// TwinCAT 3 PLC project SFICrane
// ProgramVersion: 3.1.4023.0
// libraries:
//   Tc2_MC2, * (Beckhoff Automation GmbH)
//   Tc2_MC2_Drive, * (Beckhoff Automation GmbH)
//   Tc2_Standard, * (Beckhoff Automation GmbH)
//   Tc2_System, * (Beckhoff Automation GmbH)
//   Tc2_Utilities, * (Beckhoff Automation GmbH)
//   Tc3_Module, * (Beckhoff Automation GmbH)
// project tree:
//   AXIS CONTROL/ GVL_AXIS1.TcGVL, GVL_AXIS2.TcGVL (not stored), GVL_AXIS3.TcGVL, GVL_AXIS4.TcGVL (not stored), GVL_Safety_AXIS4.TcGVL (not stored), GVL_Safety_IO.TcGVL, P_AxisControl.TcPOU, ST_MC_CMD.TcDUT, ST_MC_ParametersAxis.TcDUT, ST_MC_Status.TcDUT (not stored)
//   INPUTS/Function Blocks/ FB_AnalogInputScaling.TcPOU, FB_JoystickInputScaling.TcPOU
//   INPUTS/ G_Inputs.TcGVL, G_Sensors.TcGVL (not stored), P_Inputs.TcPOU (not stored)
//   INPUTS/Struct/ ST_AnalogInput.TcDUT (not stored), ST_AnalogInputScaling.TcDUT (not stored), ST_AnalogInputStatus.TcDUT, ST_JoystickInputScaling.TcDUT (not stored)
//   MACHINE CONTROL/ G_Parameters.TcGVL, G_Work.TcGVL (not stored), P_MachineControl.TcPOU
//   MACHINE CONTROL/InverseKinematics2d/ cosd.TcPOU (not stored), FB_InverseKin2d.TcPOU (not stored), GVL_InverseKinematics.TcGVL (not stored), rt_ceild.TcPOU (not stored), rt_floord.TcPOU, rt_remd.TcPOU (not stored)
//   MACHINE CONTROL/Struct/ ST_Parameters.TcDUT (not stored)
//   OUTPUTS/ G_Outputs.TcGVL (not stored), P_Outputs.TcPOU (not stored)
//   / PlcTask.TcTTO
//   POUs/ MAIN.TcPOU
// real-time tasks:
//   TASK PlcTask: cycle T#10ms, priority 20, ADS port 350
// motion (NC):
//   TASK NC-Task 1 SAF: cycle T#2ms, priority 4, ADS port 501
//   TASK NC-Task 1 SVB: cycle T#10ms, priority 8, ADS port 511
//   AXIS Axis 1 - Bottom cylinder (id 1)
//     OtherSettings: AllowMotionCmdToSlave=true
//     encoder EncType=8
//       EncPara: MaxCount=#x0036ee7f
//     drive DrvType=9
//       DrvPara: MaxCount=#xffffffff, DriveControlDWord=#x00030000
//         Analog: VeloScale=6, TorqueSetpointScale=10, ScaleFactorActTorque=0.1
//         TimeComp: TaskDelayCycles=1
//     controller CtrType=1
//       CtrPara: PriorControlFactor=1
//         Observer: BandWidth=20
//   AXIS Axis 2 - Slew motor (id 2)
//     OtherSettings: AllowMotionCmdToSlave=true
//     encoder EncType=8
//       EncPara: MaxCount=#x0036ee7f
//     drive DrvType=9
//       DrvPara: MaxCount=#xffffffff, DriveControlDWord=#x00030000
//         Analog: VeloScale=6, TorqueSetpointScale=10, ScaleFactorActTorque=0.1
//         TimeComp: TaskDelayCycles=1
//     controller CtrType=1
//       CtrPara: PriorControlFactor=1
//         Observer: BandWidth=20
//   AXIS Axis 3 - Top cylinder (id 3)
//     OtherSettings: AllowMotionCmdToSlave=true
//     encoder EncType=8
//       EncPara: MaxCount=#x0036ee7f
//     drive DrvType=9
//       DrvPara: MaxCount=#xffffffff, DriveControlDWord=#x00030000
//         Analog: VeloScale=6, TorqueSetpointScale=10, ScaleFactorActTorque=0.1
//         TimeComp: TaskDelayCycles=1
//     controller CtrType=1
//       CtrPara: PriorControlFactor=1
//         Observer: BandWidth=20
//   AXIS Axis 4 - Winch motor (id 4)
//     OtherSettings: AllowMotionCmdToSlave=true
//     encoder EncType=19
//       EncPara: MaxCount=#xffffffff
//     drive DrvType=16
//       DrvPara: MaxCount=#xffffffff, DriveControlDWord=#x00020100
//         Analog: TorqueSetpointScale=10, ScaleFactorActTorque=0.1
//         TimeComp: TaskDelayCycles=1
//     controller CtrType=1
//       CtrPara: PriorControlFactor=1
//         Observer: BandWidth=20
// I/O:
//   DEVICE Device 1 (EtherCAT), AmsNetId 5.107.189.26.2.1
//     Term 1 (EK1200) [EK1200-5000 EtherCAT Power supply (2A E-Bus)]
//       Term 2 (EL6910) [EL6910, TwinSAFE PLC]
//       Term 3 (EK1110) [EK1110 EtherCAT extension]
//     Term 4 (EK1818) [EK1818 EtherCAT IO-Coupler  (1A E-Bus, 8 Ch. Dig. In, 3ms, 4 Ch. Dig. Out 24V, 0,5A)]
//       Term 5 (EL3255) [EL3255 5Ch. potentiometer measurement with sensor supply]
//       Term 7 (EL9011) [EL9011 End Terminal]
//     Box 6 (AMI8000-0100) [AMI8000-0100 Servo motor 48 V DC, TwinSAFE]
//       modules: Module 1 (SAFETY)
//   DEVICE Device 4 (EtherCAT), AmsNetId 5.107.189.26.5.1
//     Drive 8 (IndraDrive MPB16/17) [IndraDrive MPB16/17]
//     Drive 9 (IndraDrive MPB20/21) [IndraDrive MPB20/21]
//     Drive 10 (IndraDrive MPB20/21) [IndraDrive MPB20/21]
// variable links:
//   NC-Task 1 SAF/Axes/Axis 1 - Bottom cylinder <-> Device 4 (EtherCAT)/Drive 8 (IndraDrive MPB16/17)
//     Drive/Inputs/In/nDcOutputTime <-> InfoData/DcOutputShift
//     Drive/Inputs/In/nState1 <-> AT/Drive status word @bit 8
//     Drive/Inputs/In/nState2 <-> AT/Drive status word
//     Drive/Inputs/In/nState4 @bit 1 <-> WcState/InputToggle
//     Drive/Inputs/In/nState4 <-> WcState/WcState
//     Drive/Outputs/Out/nCtrl1 <-> MDT/Master control word @bit 8
//     Drive/Outputs/Out/nDataOut1 <-> MDT/Position command value
//     Enc/Inputs/In/nDataIn1 <-> AT/Position feedback value 1
//     Enc/Inputs/In/nDcInputTime <-> InfoData/DcInputShift
//     Enc/Inputs/In/nState4 @bit 1 <-> WcState/InputToggle
//     Enc/Inputs/In/nState4 <-> WcState/WcState
//   NC-Task 1 SAF/Axes/Axis 2 - Slew motor <-> Device 4 (EtherCAT)/Drive 9 (IndraDrive MPB20/21)
//     Drive/Inputs/In/nDcOutputTime <-> InfoData/DcOutputShift
//     Drive/Inputs/In/nState1 <-> AT/Drive status word @bit 8
//     Drive/Inputs/In/nState2 <-> AT/Drive status word
//     Drive/Inputs/In/nState4 @bit 1 <-> WcState/InputToggle
//     Drive/Inputs/In/nState4 <-> WcState/WcState
//     Drive/Outputs/Out/nCtrl1 <-> MDT/Master control word @bit 8
//     Drive/Outputs/Out/nDataOut1 <-> MDT/Position command value
//     Enc/Inputs/In/nDataIn1 <-> AT/Position feedback value 1
//     Enc/Inputs/In/nDcInputTime <-> InfoData/DcInputShift
//     Enc/Inputs/In/nState4 @bit 1 <-> WcState/InputToggle
//     Enc/Inputs/In/nState4 <-> WcState/WcState
//   NC-Task 1 SAF/Axes/Axis 3 - Top cylinder <-> Device 4 (EtherCAT)/Drive 10 (IndraDrive MPB20/21)
//     Drive/Inputs/In/nDcOutputTime <-> InfoData/DcOutputShift
//     Drive/Inputs/In/nState1 <-> AT/Drive status word @bit 8
//     Drive/Inputs/In/nState2 <-> AT/Drive status word
//     Drive/Inputs/In/nState4 @bit 1 <-> WcState/InputToggle
//     Drive/Inputs/In/nState4 <-> WcState/WcState
//     Drive/Outputs/Out/nCtrl1 <-> MDT/Master control word @bit 8
//     Drive/Outputs/Out/nDataOut1 <-> MDT/Position command value
//     Enc/Inputs/In/nDataIn1 <-> AT/Position feedback value 1
//     Enc/Inputs/In/nDcInputTime <-> InfoData/DcInputShift
//     Enc/Inputs/In/nState4 @bit 1 <-> WcState/InputToggle
//     Enc/Inputs/In/nState4 <-> WcState/WcState
//   NC-Task 1 SAF/Axes/Axis 4 - Winch motor <-> Device 1 (EtherCAT)/Box 6 (AMI8000-0100)
//     Drive/Inputs/In/nDataIn1 <-> DRV Following error actual value/Following error actual value
//     Drive/Inputs/In/nDcOutputTime <-> InfoData/DcOutputShift
//     Drive/Inputs/In/nState1 <-> DRV Statusword/Statusword
//     Drive/Inputs/In/nState2 <-> DRV Statusword/Statusword @bit 8
//     Drive/Inputs/In/nState4 @bit 1 <-> WcState/InputToggle
//     Drive/Inputs/In/nState4 <-> WcState/WcState
//     Drive/Outputs/Out/nCtrl1 <-> DRV Controlword/Controlword
//     Drive/Outputs/Out/nCtrl2 <-> DRV Controlword/Controlword @bit 8
//     Drive/Outputs/Out/nDataOut1 <-> DRV Target position/Target position
//     Enc/Inputs/In/nDataIn1 <-> FB Position/Position
//     Enc/Inputs/In/nDcInputTime <-> InfoData/DcInputShift
//     Enc/Inputs/In/nState4 @bit 1 <-> WcState/InputToggle
//     Enc/Inputs/In/nState4 <-> WcState/WcState
//   SFICrane/SFICrane Instance <-> Device 1 (EtherCAT)/Term 4 (EK1818)
//     PlcTask Inputs/G_Inputs.bAutoModeSelector <-> Channel 4/Input
//     PlcTask Inputs/G_Inputs.bGreenButton <-> Channel 5/Input
//     PlcTask Inputs/G_Inputs.bJoystickLeftEnable <-> Channel 7/Input
//     PlcTask Inputs/G_Inputs.bJoystickRightEnable <-> Channel 8/Input
//     PlcTask Inputs/G_Inputs.bManualModeSelector <-> Channel 3/Input
//     PlcTask Inputs/G_Inputs.bRedButton <-> Channel 6/Input
//     PlcTask Outputs/G_Outputs.bGreenButtonLight <-> Channel 9/Output
//     PlcTask Outputs/G_Outputs.bRedButtonLight <-> Channel 10/Output
//   SFICrane/SFICrane Instance <-> Device 1 (EtherCAT)/Term 4 (EK1818)/Term 5 (EL3255)
//     PlcTask Inputs/G_Inputs.stJoyLX.nValue <-> AI Standard Channel 1/Value
//     PlcTask Inputs/G_Inputs.stJoyLX.stStatus <-> AI Standard Channel 1/Status
//     PlcTask Inputs/G_Inputs.stJoyLY.nValue <-> AI Standard Channel 2/Value
//     PlcTask Inputs/G_Inputs.stJoyLY.stStatus <-> AI Standard Channel 2/Status
//     PlcTask Inputs/G_Inputs.stJoyRX.nValue <-> AI Standard Channel 3/Value
//     PlcTask Inputs/G_Inputs.stJoyRX.stStatus <-> AI Standard Channel 3/Status
//     PlcTask Inputs/G_Inputs.stJoyRY.nValue <-> AI Standard Channel 4/Value
//     PlcTask Inputs/G_Inputs.stJoyRY.stStatus <-> AI Standard Channel 4/Status
//   SFICrane/SFICrane Instance <-> NC-Task 1 SAF/Axes/Axis 1 - Bottom cylinder
//     PlcTask Inputs/GVL_AXIS1.BCAxis.NcToPlc <-> Outputs/ToPlc
//     PlcTask Outputs/GVL_AXIS1.BCAxis.PlcToNc <-> Inputs/FromPlc
//   SFICrane/SFICrane Instance <-> NC-Task 1 SAF/Axes/Axis 2 - Slew motor
//     PlcTask Inputs/GVL_AXIS2.SJAxis.NcToPlc <-> Outputs/ToPlc
//     PlcTask Outputs/GVL_AXIS2.SJAxis.PlcToNc <-> Inputs/FromPlc
//   SFICrane/SFICrane Instance <-> NC-Task 1 SAF/Axes/Axis 3 - Top cylinder
//     PlcTask Inputs/GVL_AXIS3.TCAxis.NcToPlc <-> Outputs/ToPlc
//     PlcTask Outputs/GVL_AXIS3.TCAxis.PlcToNc <-> Inputs/FromPlc
//   SFICrane/SFICrane Instance <-> NC-Task 1 SAF/Axes/Axis 4 - Winch motor
//     PlcTask Inputs/GVL_AXIS4.WMAxis.NcToPlc <-> Outputs/ToPlc
//     PlcTask Outputs/GVL_AXIS4.WMAxis.PlcToNc <-> Inputs/FromPlc

CONFIGURATION SFICrane
    RESOURCE PLC ON TwinCAT3
        TASK PlcTask(INTERVAL := T#10ms, PRIORITY := 20);
        PROGRAM MAIN WITH PlcTask : MAIN;
    END_RESOURCE
END_CONFIGURATION

// ---- AXIS CONTROL/ST_MC_CMD.TcDUT
TYPE ST_MC_CMD :
STRUCT
	
bExe				: BOOL;
lrVelocity			: LREAL;
lrAcceleration		: LREAL;
lrDeceleration		: LREAL;
lrJerk				: LREAL;
lrDistance			: LREAL;
lrPosition			: LREAL;
EnuDirection		: MC_Direction;
EnuBufferMode		: MC_BufferMode;
EnuOptions			: ST_MoveOptions;

END_STRUCT
END_TYPE

// ---- AXIS CONTROL/ST_MC_ParametersAxis.TcDUT
TYPE ST_MC_ParametersAxis :
STRUCT
	
	

END_STRUCT
END_TYPE

// ---- INPUTS/Struct/ST_AnalogInputStatus.TcDUT
TYPE ST_AnalogInputStatus :
STRUCT
	Underrange 		: BIT; // 0.0
	Overrange 		: BIT; // 0.1
	Limit_1_0 		: BIT; // 0.2
	Limit_1_1 		: BIT; // 0.3
	Limit_2_0 		: BIT; // 0.4
	Limit_2_1 		: BIT; // 0.5
	Error 			: BIT; // 0.6
	Reserved_0_7	: BIT; // 0.7
	Reserved_1_0 	: BIT; // 1.0
	Reserved_1_1 	: BIT; // 1.1
	Reserved_1_2 	: BIT; // 1.2
	Reserved_1_3 	: BIT; // 1.3
	Reserved_1_4 	: BIT; // 1.4
	Reserved_1_5 	: BIT; // 1.5
	TxPDO_State 	: BIT; // 1.6
	TxPDO_Toggle 	: BIT; // 1.7	
END_STRUCT
END_TYPE

// ---- AXIS CONTROL/GVL_AXIS1.TcGVL
{attribute 'qualified_only'}
VAR_GLOBAL

//Axis1 Bottom Cylinder 'BC'
BCAxis : AXIS_REF;

//Motion Control Function Block Instant Variable 
fbBC_Reset				: MC_Reset;
fbBC_Power				: MC_Power;
fbBC_Home				: MC_Home;
fbBC_Jog				: MC_Jog;
fbBC_MoveVelocity		: MC_MoveVelocity;
fbBC_Stop				: MC_Stop;
fbBC_MoveAbs			: MC_MoveAbsolute;
fbBC_MoveContAbs		: MC_MoveContinuousAbsolute;
fbBC_SetPosition		: MC_SetPosition;
fbBC_MoveAdditive		: MC_MoveAdditive;

//Input: Command
bBC_ResetExe			: BOOL;

bBC_PowerEnCmd			: BOOL;
bBC_PowerEnPositive		: BOOL;
bBC_PowerEnNegative 	: BOOL;

bBC_HomeExe				: BOOL;
bBC_HomeCamInput		: BOOL;

bBC_JogFwd				: BOOL;
bBC_JogRev				: BOOL;	

bBC_MoveVelExe			: BOOL;
	
bBC_StopExe				: BOOL;

bBC_MoveAbsExe			: BOOL;

bBC_MoveContAbsExe		: BOOL;

bBC_MoveContAbsInEndVel	: BOOL;

bBC_MoveAddExe			: BOOL;


fBC_MoveContAbsExeTrig	: UINT;


stBC_VelCmd				: ST_MC_CMD := (bExe := FALSE, lrVelocity := 100, EnuDirection := MC_Positive_Direction); 
//stBC_VelCmd				: ST_MC_CMD := (bExe := FALSE, lrVelocity := 100, lrAcceleration := 0, lrDeceleration := 0, lrJerk := 0, lrDistance := 0, lrPosition := 0, EnuDirection := MC_Positive_Direction, EnuBufferMode := 0, EnuOptions := 0 ); 

//Variables/Parameters
lrBC_PowerOverride		: LREAL;
lrBC_HomePosition		: LREAL;
lrBC_JogVelocity		: LREAL;
lrBC_MoveVelVelocity	: LREAL;
lrBC_MoveAbsPosition	: LREAL;
lrBC_MoveContAbsPos		: LREAL;
lrBC_MoveContAbsEndVel 	: LREAL := 0;
lrBC_MoveAddPos		: LREAL;

//Direction
EnuMoveVelDirection		: MC_Direction;

// Status
stBC_Reset				: ST_MC_Status;
stBC_Power				: ST_MC_Status;
stBC_Home				: ST_MC_Status;
stBC_Jog				: ST_MC_Status;
stBC_MoveVelocity		: ST_MC_Status;
stBC_Stop				: ST_MC_Status;
stBC_MoveAbs			: ST_MC_Status;
stBC_MoveContAbs		: ST_MC_Status;
stBC_MoveAdd			: ST_MC_Status;

END_VAR

// ---- AXIS CONTROL/GVL_AXIS3.TcGVL
{attribute 'qualified_only'}
VAR_GLOBAL

//Axis3 Top Cylinder 'TC'
TCAxis : AXIS_REF;

//Motion Control Function Block Instant Variable 
fbTC_Reset				: MC_Reset;
fbTC_Power				: MC_Power;
fbTC_Home				: MC_Home;
fbTC_Jog				: MC_Jog;
fbTC_MoveVelocity		: MC_MoveVelocity;
fbTC_Stop				: MC_Stop;
fbTC_MoveAbs			: MC_MoveAbsolute;

//Input: Command
bTC_ResetExe			: BOOL;

bTC_PowerEnCmd			: BOOL;
bTC_PowerEnPositive		: BOOL;
bTC_PowerEnNegative 	: BOOL;

bTC_HomeExe				: BOOL;
bTC_HomeCamInput		: BOOL;

bTC_JogFwd				: BOOL;
bTC_JogRev				: BOOL;	

bTC_MoveVelExe			: BOOL;
	
bTC_StopExe				: BOOL;

bTC_MoveAbsExe			: BOOL;

stTC_VelCmd				: ST_MC_CMD := (bExe := FALSE, lrVelocity := 100, EnuDirection := MC_Positive_Direction); 
//stTC_VelCmd				: ST_MC_CMD := (bExe := FALSE, lrVelocity := 100, lrAcceleration := 0, lrDeceleration := 0, lrJerk := 0, lrDistance := 0, lrPosition := 0, EnuDirection := MC_Positive_Direction, EnuBufferMode := 0, EnuOptions := 0 ); 

//Variables/Parameters
lrTC_PowerOverride		: LREAL;
lrTC_HomePosition		: LREAL;
lrTC_SetPosition		: LREAL;
lrTC_JogVelocity		: LREAL;
lrTC_MoveVelVelocity	: LREAL;
lrTC_MoveAbsPosition	: LREAL;

//Direction
EnuMoveVelDirection		: MC_Direction;

// Status
stTC_Reset				: ST_MC_Status;
stTC_Power				: ST_MC_Status;
stTC_Home				: ST_MC_Status;
stTC_SetPosition		: ST_MC_Status;
stTC_Jog				: ST_MC_Status;
stTC_MoveVelocity		: ST_MC_Status;
stTC_Stop				: ST_MC_Status;
stTC_MoveAbs			: ST_MC_Status;

END_VAR

// ---- AXIS CONTROL/GVL_Safety_IO.TcGVL
{attribute 'qualified_only'}
VAR_GLOBAL
	bInAckSignal		AT %I* 	: BOOL := TRUE;
	bEStop				AT %I*	: BOOL := FALSE;
END_VAR

// ---- INPUTS/G_Inputs.TcGVL
{attribute 'qualified_only'}
VAR_GLOBAL
	bManualModeSelector			AT %I* : BOOL;
	bAutoModeSelector			AT %I* : BOOL;
	bRedButton					AT %I* : BOOL;
	bGreenButton				AT %I* : BOOL;
	bJoystickLeftEnable			AT %I* : BOOL;
	bJoystickRightEnable		AT %I* : BOOL;
	
	// Analog Inputs
	stJoyLX 					: ST_AnalogInput;
	stJoyLY						: ST_AnalogInput;
	stJoyRX 					: ST_AnalogInput;
	stJoyRY						: ST_AnalogInput;

END_VAR

// ---- MACHINE CONTROL/G_Parameters.TcGVL
{attribute 'qualified_only'}
VAR_GLOBAL
	stParam : ST_Parameters;
END_VAR

// ---- POUs/MAIN.TcPOU
PROGRAM MAIN

VAR
bEnable: BOOL := FALSE;
bMove: BOOL := FALSE;
fAxis1VelocityPercent: LREAL := 0;	
axis1: AXIS_REF;
fbAxis1Power: MC_Power;
fbAxis1MoveVelocity: MC_MoveVelocity;
MCDirectionAxis1 : MC_Direction;
fAxis1ReferenceVelocity: LREAL := 100;
END_VAR

P_Inputs();
P_MachineControl();
P_AxisControl();
P_Outputs();

(*

bEnable := G_Inputs.bJoystickLeftEnable;
bMove := G_Inputs.bJoystickLeftEnable;
fAxis1VelocityPercent := ABS(G_Sensors.fJoystickLeftNormalizedX)*100;
MCDirectionAxis1 := G_Sensors.MCDirectionAxis1;

axis1.ReadStatus();

fbAxis1Power(
Axis:= axis1,
Enable:= bEnable,
Enable_Positive:= bEnable,
Enable_Negative:= bEnable,
Override:= fAxis1VelocityPercent,
BufferMode:= ,
Options:= ,
Status=> ,
Busy=> ,
Active=> ,
Error=> ,
ErrorID=> );

fbAxis1MoveVelocity(
Axis:= axis1,
Execute:= bMove,
Velocity:= fAxis1ReferenceVelocity,
Acceleration:= ,
Deceleration:= ,
Jerk:= ,
Direction:= G_Sensors.MCDirectionAxis1,
BufferMode:= ,
Options:= ,
InVelocity=> ,
Busy=> ,
Active=> ,
CommandAborted=> ,
Error=> ,
ErrorID=> );

*)

END_PROGRAM

// ---- MACHINE CONTROL/P_MachineControl.TcPOU
PROGRAM P_MachineControl
VAR
	fbInverse					: FB_InverseKin2d;
	fRefPosX					: LREAL := GVL_InverseKinematics.fTooltipXCoordGlobalIni;
	fRefPosY					: LREAL := GVL_InverseKinematics.fTooltipYCoordGlobalIni;					
END_VAR

G_Work.bManualMode := G_Inputs.bManualModeSelector;
G_Work.bAutoMode := G_Inputs.bAutoModeSelector;

IF G_Inputs.bAutoModeSelector THEN
fRefPosX := fRefPosX + G_Sensors.fJoystickLeftNormalizedX*-0.001;
fRefPosY := fRefPosY + G_Sensors.fJoystickLeftNormalizedY*0.001;
END_IF

fbInverse(
	fPtXd := fRefPosX, 
	fPtYd := fRefPosY, 
	fTheta1 :=GVL_InverseKinematics.fTheta1,
	
	fTheta3 => GVL_InverseKinematics.fAngleMainArmInverse, 
	fTheta4 => GVL_InverseKinematics.fAngleKnuckleArmInverse,
	fStrokeActuatorMain => GVL_InverseKinematics.fStrokeActuatorMainInverse,
	fStrokeActuatorKnuckle => GVL_InverseKinematics.fStrokeActuatorKnuckleInverse,	
);

END_PROGRAM

// ---- AXIS CONTROL/P_AxisControl.TcPOU
PROGRAM P_AxisControl
VAR
END_VAR

//Axis Control program based on youtube series Twincat 3 NC Videos MB05a until MB17b plus MB22 by @electricalautomation https://www.youtube.com/watch?v=BxRAOdTks9I&list=PL762SfoJC-e8NbAUQ-H7a_TOdqrlBPCw4&index=25

AXIS1_LD();

GVL_AXIS1.bBC_ResetExe := G_Inputs.bJoystickLeftEnable OR G_Inputs.bAutoModeSelector;

GVL_AXIS1.EnuMoveVelDirection := G_Sensors.MCDirectionAxis1;

GVL_AXIS1.bBC_PowerEnCmd := G_Inputs.bManualModeSelector OR G_Inputs.bAutoModeSelector;
GVL_AXIS1.bBC_PowerEnNegative := G_Inputs.bManualModeSelector OR G_Inputs.bAutoModeSelector;
GVL_AXIS1.bBC_PowerEnPositive := G_Inputs.bManualModeSelector OR G_Inputs.bAutoModeSelector;

GVL_AXIS1.lrBC_JogVelocity := 100;
GVL_AXIS1.lrBC_PowerOverride := 50;

GVL_AXIS1.lrBC_MoveAddPos := GVL_InverseKinematics.fStrokeActuatorMainInverse*1000; //Position in mm

GVL_AXIS1.lrBC_MoveContAbsEndVel := 0;

// Jog control

(*
IF G_Sensors.fJoystickLeftNormalizedX  > 0 AND G_Inputs.bJoystickLeftEnable THEN
	GVL_AXIS1.bBC_JogRev := TRUE;
ELSIF G_Sensors.fJoystickLeftNormalizedX < 0 AND G_Inputs.bJoystickLeftEnable THEN
	GVL_AXIS1.bBC_JogFwd := TRUE;
ELSE
	 GVL_AXIS1.bBC_JogFwd := FALSE;
	 GVL_AXIS1.bBC_JogRev := FALSE;
END_IF

*)



// Manual velocity control
IF G_Sensors.fJoystickLeftNormalizedX  >= 0 AND G_Inputs.bJoystickLeftEnable AND G_Inputs.bManualModeSelector THEN
	GVL_AXIS1.lrBC_PowerOverride := ABS(G_Sensors.fJoystickLeftNormalizedX) * 100;
	GVL_AXIS1.stBC_VelCmd.EnuDirection := MC_Positive_Direction;
	GVL_AXIS1.stBC_VelCmd.bExe := TRUE;
	GVL_AXIS1.bBC_StopExe := FALSE;
ELSIF G_Sensors.fJoystickLeftNormalizedX < 0 AND G_Inputs.bJoystickLeftEnable AND G_Inputs.bManualModeSelector THEN
	GVL_AXIS1.lrBC_PowerOverride := ABS(G_Sensors.fJoystickLeftNormalizedX) * 100;
	GVL_AXIS1.stBC_VelCmd.EnuDirection := MC_Negative_Direction;
	GVL_AXIS1.stBC_VelCmd.bExe := TRUE;
	GVL_AXIS1.bBC_StopExe := FALSE;
ELSIF G_Inputs.bAutoModeSelector THEN
	GVL_AXIS1.lrBC_PowerOverride := 20;
	GVL_AXIS1.bBC_StopExe := FALSE;
	//GVL_AXIS1.stBC_VelCmd.EnuDirection := MC_Positive_Direction;
	//GVL_AXIS1.stBC_VelCmd.bExe := TRUE;
	//GVL_AXIS1.bBC_MoveAddExe := TRUE;
ELSE
	 GVL_AXIS1.lrBC_PowerOverride := 0;
	 //GVL_AXIS1.stBC_VelCmd.EnuDirection := MC_Current_Direction;
	 GVL_AXIS1.stBC_VelCmd.bExe := FALSE;
	 //GVL_AXIS1.bBC_StopExe := TRUE;
END_IF

IF GVL_AXIS1.stBC_MoveAdd.Done THEN
	GVL_AXIS1.bBC_MoveAddExe := FALSE;
END_IF

(*
// Automatic position control

IF G_Inputs.bAutoModeSelector THEN
	GVL_AXIS1.lrBC_PowerOverride := 10;
	//GVL_AXIS1.stBC_VelCmd.EnuDirection := MC_Positive_Direction;
	GVL_AXIS1.stBC_VelCmd.bExe := TRUE;
	GVL_AXIS1.bBC_MoveAbsExe := TRUE;
ELSE
	 GVL_AXIS1.lrBC_PowerOverride := 0;
	 //GVL_AXIS1.stBC_VelCmd.EnuDirection := MC_Current_Direction;
	 GVL_AXIS1.stBC_VelCmd.bExe := FALSE;
END_IF
*)

AXIS2_LD();

GVL_AXIS2.bSJ_ResetExe := G_Inputs.bJoystickRightEnable;

GVL_AXIS2.EnuMoveVelDirection := G_Sensors.MCDirectionAxis2;

GVL_AXIS2.bSJ_PowerEnCmd := G_Inputs.bManualModeSelector;
GVL_AXIS2.bSJ_PowerEnNegative := G_Inputs.bManualModeSelector;
GVL_AXIS2.bSJ_PowerEnPositive := G_Inputs.bManualModeSelector;

GVL_AXIS2.lrSJ_JogVelocity := 100;


// Velocity control
IF G_Sensors.fJoystickRightNormalizedX  > 0 AND G_Inputs.bJoystickRightEnable THEN
	GVL_AXIS2.lrSJ_PowerOverride := ABS(G_Sensors.fJoystickRightNormalizedX) * 100;
	GVL_AXIS2.stSJ_VelCmd.EnuDirection := MC_Positive_Direction;
	GVL_AXIS2.stSJ_VelCmd.bExe := TRUE;
ELSIF G_Sensors.fJoystickRightNormalizedX < 0 AND G_Inputs.bJoystickRightEnable THEN
	GVL_AXIS2.lrSJ_PowerOverride := ABS(G_Sensors.fJoystickRightNormalizedX) * 100;
	GVL_AXIS2.stSJ_VelCmd.EnuDirection := MC_Negative_Direction;
	GVL_AXIS2.stSJ_VelCmd.bExe := TRUE;
ELSE
	 GVL_AXIS2.lrSJ_PowerOverride := 0;
	 //GVL_AXIS2.stSJ_VelCmd.EnuDirection := MC_Current_Direction;
	 GVL_AXIS2.stSJ_VelCmd.bExe := FALSE;
END_IF


AXIS3_LD();

GVL_AXIS3.bTC_ResetExe := G_Inputs.bJoystickLeftEnable;

GVL_AXIS3.EnuMoveVelDirection := G_Sensors.MCDirectionAxis3;

GVL_AXIS3.bTC_PowerEnCmd := G_Inputs.bManualModeSelector;
GVL_AXIS3.bTC_PowerEnNegative := G_Inputs.bManualModeSelector;
GVL_AXIS3.bTC_PowerEnPositive := G_Inputs.bManualModeSelector;

GVL_AXIS3.lrTC_JogVelocity := 100;


// Velocity control
IF G_Sensors.fJoystickLeftNormalizedY  > 0 AND G_Inputs.bJoystickLeftEnable THEN
	GVL_AXIS3.lrTC_PowerOverride := ABS(G_Sensors.fJoystickLeftNormalizedY) * 100;
	GVL_AXIS3.stTC_VelCmd.EnuDirection := MC_Positive_Direction;
	GVL_AXIS3.stTC_VelCmd.bExe := TRUE;
ELSIF G_Sensors.fJoystickLeftNormalizedY < 0 AND G_Inputs.bJoystickLeftEnable THEN
	GVL_AXIS3.lrTC_PowerOverride := ABS(G_Sensors.fJoystickLeftNormalizedY) * 100;
	GVL_AXIS3.stTC_VelCmd.EnuDirection := MC_Negative_Direction;
	GVL_AXIS3.stTC_VelCmd.bExe := TRUE;
ELSE
	 GVL_AXIS3.lrTC_PowerOverride := 0;
	 //GVL_AXIS3.stTC_VelCmd.EnuDirection := MC_Current_Direction;
	 GVL_AXIS3.stTC_VelCmd.bExe := FALSE;
END_IF

(*
AXIS4_LD();

//Safety
GVL_Safety_AXIS4.bSafetyRestart := GVL_AXIS4.bInAckSignal;
GVL_Safety_AXIS4.bErrorAck		:= GVL_AXIS4.bInAckSignal;
GVL_Safety_AXIS4.bSafetyRun		:= TRUE;

//
GVL_AXIS4.bWM_ResetExe := G_Inputs.bJoystickLeftEnable;

GVL_AXIS4.EnuMoveVelDirection := G_Sensors.MCDirectionAxis4;

GVL_AXIS4.bWM_PowerEnCmd := G_Inputs.bManualModeSelector;
GVL_AXIS4.bWM_PowerEnNegative := G_Inputs.bManualModeSelector;
GVL_AXIS4.bWM_PowerEnPositive := G_Inputs.bManualModeSelector;

GVL_AXIS4.lrWM_JogVelocity := 100;
//GVL_AXIS4.lrWM_PowerOverride := 50;


// Velocity control
IF G_Sensors.fJoystickLeftNormalizedY  > 0 AND G_Inputs.bJoystickLeftEnable THEN
	GVL_AXIS4.lrWM_PowerOverride := ABS(G_Sensors.fJoystickLeftNormalizedY) * 100;
	GVL_AXIS4.stWM_VelCmd.EnuDirection := MC_Positive_Direction;
	GVL_AXIS4.stWM_VelCmd.bExe := TRUE;
ELSIF G_Sensors.fJoystickLeftNormalizedY < 0 AND G_Inputs.bJoystickLeftEnable THEN
	GVL_AXIS4.lrWM_PowerOverride := ABS(G_Sensors.fJoystickLeftNormalizedY) * 100;
	GVL_AXIS4.stWM_VelCmd.EnuDirection := MC_Negative_Direction;
	GVL_AXIS4.stWM_VelCmd.bExe := TRUE;
ELSE
	 GVL_AXIS4.lrWM_PowerOverride := 0;
	 GVL_AXIS4.stWM_VelCmd.EnuDirection := MC_Current_Direction;
	 GVL_AXIS4.stWM_VelCmd.bExe := FALSE;
END_IF
*)

METHOD AXIS1_LD : BOOL
VAR_INPUT
END_VAR
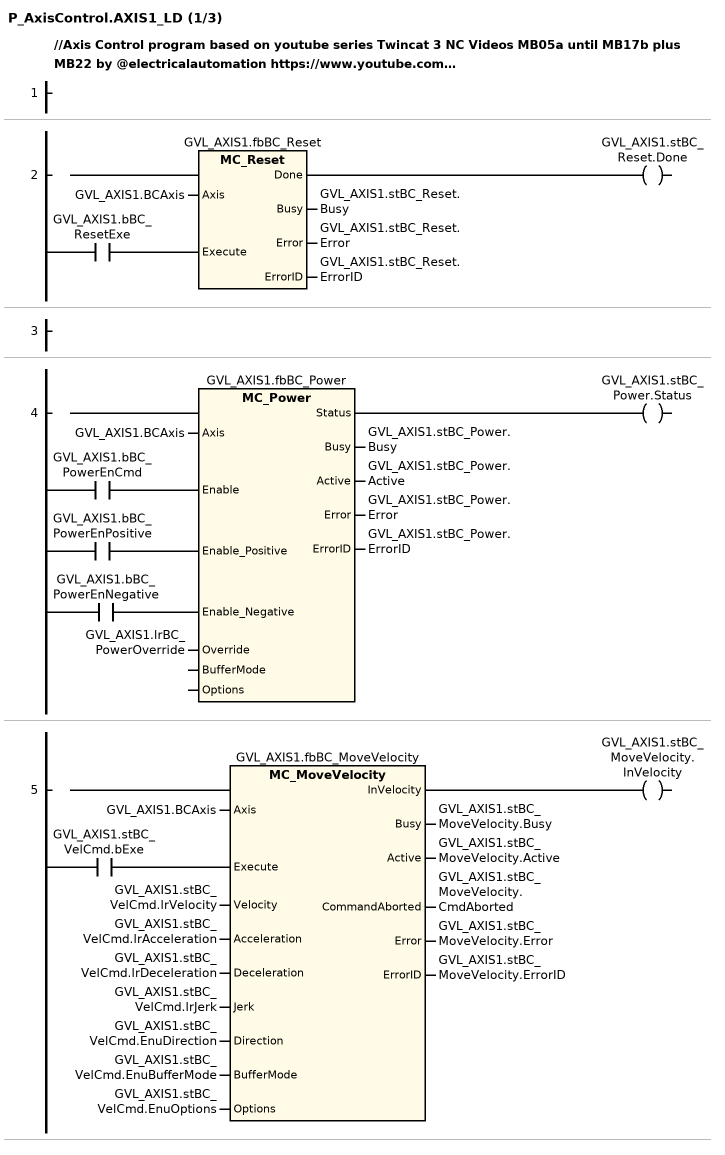
// NETWORK 1: //Axis Control program based on youtube series Twincat 3 NC Videos MB05a until MB17b plus MB22 by @electricalautomation https://www.youtube.com/watch?v=BxRAOdTks9I&list=PL762SfoJC-e8NbAUQ-H7a_TOdqrlBPCw4&index=25

// NETWORK 2
GVL_AXIS1.fbBC_Reset(
    Axis := GVL_AXIS1.BCAxis,
    Execute := GVL_AXIS1.bBC_ResetExe,
    Busy => GVL_AXIS1.stBC_Reset.Busy,
    Error => GVL_AXIS1.stBC_Reset.Error,
    ErrorID => GVL_AXIS1.stBC_Reset.ErrorID); // MC_Reset
GVL_AXIS1.stBC_Reset.Done := GVL_AXIS1.fbBC_Reset.Done;

// NETWORK 3

// NETWORK 4
GVL_AXIS1.fbBC_Power(
    Axis := GVL_AXIS1.BCAxis,
    Enable := GVL_AXIS1.bBC_PowerEnCmd,
    Enable_Positive := GVL_AXIS1.bBC_PowerEnPositive,
    Enable_Negative := GVL_AXIS1.bBC_PowerEnNegative,
    Override := GVL_AXIS1.lrBC_PowerOverride,
    Busy => GVL_AXIS1.stBC_Power.Busy,
    Active => GVL_AXIS1.stBC_Power.Active,
    Error => GVL_AXIS1.stBC_Power.Error,
    ErrorID => GVL_AXIS1.stBC_Power.ErrorID); // MC_Power
GVL_AXIS1.stBC_Power.Status := GVL_AXIS1.fbBC_Power.Status;

// NETWORK 5
GVL_AXIS1.fbBC_MoveVelocity(
    Axis := GVL_AXIS1.BCAxis,
    Execute := GVL_AXIS1.stBC_VelCmd.bExe,
    Velocity := GVL_AXIS1.stBC_VelCmd.lrVelocity,
    Acceleration := GVL_AXIS1.stBC_VelCmd.lrAcceleration,
    Deceleration := GVL_AXIS1.stBC_VelCmd.lrDeceleration,
    Jerk := GVL_AXIS1.stBC_VelCmd.lrJerk,
    Direction := GVL_AXIS1.stBC_VelCmd.EnuDirection,
    BufferMode := GVL_AXIS1.stBC_VelCmd.EnuBufferMode,
    Options := GVL_AXIS1.stBC_VelCmd.EnuOptions,
    Busy => GVL_AXIS1.stBC_MoveVelocity.Busy,
    Active => GVL_AXIS1.stBC_MoveVelocity.Active,
    CommandAborted => GVL_AXIS1.stBC_MoveVelocity.CmdAborted,
    Error => GVL_AXIS1.stBC_MoveVelocity.Error,
    ErrorID => GVL_AXIS1.stBC_MoveVelocity.ErrorID); // MC_MoveVelocity
GVL_AXIS1.stBC_MoveVelocity.InVelocity := GVL_AXIS1.fbBC_MoveVelocity.InVelocity;

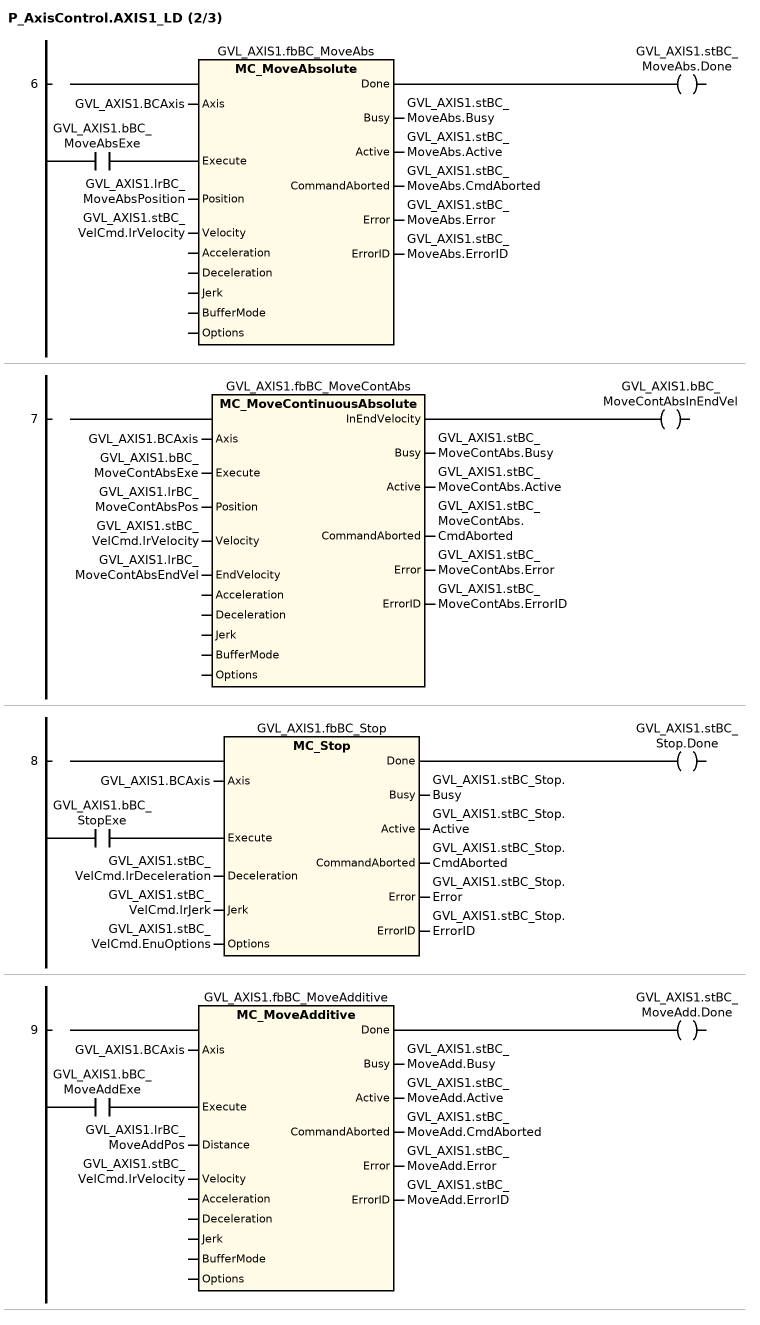
// NETWORK 6
GVL_AXIS1.fbBC_MoveAbs(
    Axis := GVL_AXIS1.BCAxis,
    Execute := GVL_AXIS1.bBC_MoveAbsExe,
    Position := GVL_AXIS1.lrBC_MoveAbsPosition,
    Velocity := GVL_AXIS1.stBC_VelCmd.lrVelocity,
    Busy => GVL_AXIS1.stBC_MoveAbs.Busy,
    Active => GVL_AXIS1.stBC_MoveAbs.Active,
    CommandAborted => GVL_AXIS1.stBC_MoveAbs.CmdAborted,
    Error => GVL_AXIS1.stBC_MoveAbs.Error,
    ErrorID => GVL_AXIS1.stBC_MoveAbs.ErrorID); // MC_MoveAbsolute
GVL_AXIS1.stBC_MoveAbs.Done := GVL_AXIS1.fbBC_MoveAbs.Done;

// NETWORK 7
GVL_AXIS1.fbBC_MoveContAbs(
    Axis := GVL_AXIS1.BCAxis,
    Execute := GVL_AXIS1.bBC_MoveContAbsExe,
    Position := GVL_AXIS1.lrBC_MoveContAbsPos,
    Velocity := GVL_AXIS1.stBC_VelCmd.lrVelocity,
    EndVelocity := GVL_AXIS1.lrBC_MoveContAbsEndVel,
    Busy => GVL_AXIS1.stBC_MoveContAbs.Busy,
    Active => GVL_AXIS1.stBC_MoveContAbs.Active,
    CommandAborted => GVL_AXIS1.stBC_MoveContAbs.CmdAborted,
    Error => GVL_AXIS1.stBC_MoveContAbs.Error,
    ErrorID => GVL_AXIS1.stBC_MoveContAbs.ErrorID); // MC_MoveContinuousAbsolute
GVL_AXIS1.bBC_MoveContAbsInEndVel := GVL_AXIS1.fbBC_MoveContAbs.InEndVelocity;

// NETWORK 8
GVL_AXIS1.fbBC_Stop(
    Axis := GVL_AXIS1.BCAxis,
    Execute := GVL_AXIS1.bBC_StopExe,
    Deceleration := GVL_AXIS1.stBC_VelCmd.lrDeceleration,
    Jerk := GVL_AXIS1.stBC_VelCmd.lrJerk,
    Options := GVL_AXIS1.stBC_VelCmd.EnuOptions,
    Busy => GVL_AXIS1.stBC_Stop.Busy,
    Active => GVL_AXIS1.stBC_Stop.Active,
    CommandAborted => GVL_AXIS1.stBC_Stop.CmdAborted,
    Error => GVL_AXIS1.stBC_Stop.Error,
    ErrorID => GVL_AXIS1.stBC_Stop.ErrorID); // MC_Stop
GVL_AXIS1.stBC_Stop.Done := GVL_AXIS1.fbBC_Stop.Done;

// NETWORK 9
GVL_AXIS1.fbBC_MoveAdditive(
    Axis := GVL_AXIS1.BCAxis,
    Execute := GVL_AXIS1.bBC_MoveAddExe,
    Distance := GVL_AXIS1.lrBC_MoveAddPos,
    Velocity := GVL_AXIS1.stBC_VelCmd.lrVelocity,
    Busy => GVL_AXIS1.stBC_MoveAdd.Busy,
    Active => GVL_AXIS1.stBC_MoveAdd.Active,
    CommandAborted => GVL_AXIS1.stBC_MoveAdd.CmdAborted,
    Error => GVL_AXIS1.stBC_MoveAdd.Error,
    ErrorID => GVL_AXIS1.stBC_MoveAdd.ErrorID); // MC_MoveAdditive
GVL_AXIS1.stBC_MoveAdd.Done := GVL_AXIS1.fbBC_MoveAdditive.Done;

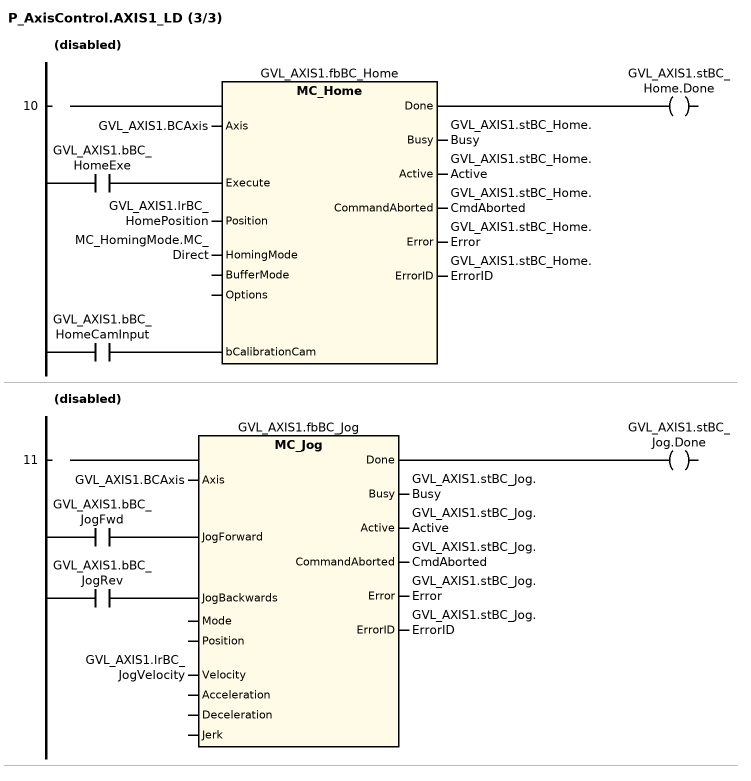
// NETWORK 10 (disabled)
// GVL_AXIS1.fbBC_Home(
//     Axis := GVL_AXIS1.BCAxis,
//     Execute := GVL_AXIS1.bBC_HomeExe,
//     Position := GVL_AXIS1.lrBC_HomePosition,
//     HomingMode := MC_HomingMode.MC_Direct,
//     bCalibrationCam := GVL_AXIS1.bBC_HomeCamInput,
//     Busy => GVL_AXIS1.stBC_Home.Busy,
//     Active => GVL_AXIS1.stBC_Home.Active,
//     CommandAborted => GVL_AXIS1.stBC_Home.CmdAborted,
//     Error => GVL_AXIS1.stBC_Home.Error,
//     ErrorID => GVL_AXIS1.stBC_Home.ErrorID); // MC_Home
// GVL_AXIS1.stBC_Home.Done := GVL_AXIS1.fbBC_Home.Done;

// NETWORK 11 (disabled)
// GVL_AXIS1.fbBC_Jog(
//     Axis := GVL_AXIS1.BCAxis,
//     JogForward := GVL_AXIS1.bBC_JogFwd,
//     JogBackwards := GVL_AXIS1.bBC_JogRev,
//     Velocity := GVL_AXIS1.lrBC_JogVelocity,
//     Busy => GVL_AXIS1.stBC_Jog.Busy,
//     Active => GVL_AXIS1.stBC_Jog.Active,
//     CommandAborted => GVL_AXIS1.stBC_Jog.CmdAborted,
//     Error => GVL_AXIS1.stBC_Jog.Error,
//     ErrorID => GVL_AXIS1.stBC_Jog.ErrorID); // MC_Jog
// GVL_AXIS1.stBC_Jog.Done := GVL_AXIS1.fbBC_Jog.Done;
END_METHOD

METHOD AXIS2_LD : BOOL
VAR_INPUT
END_VAR
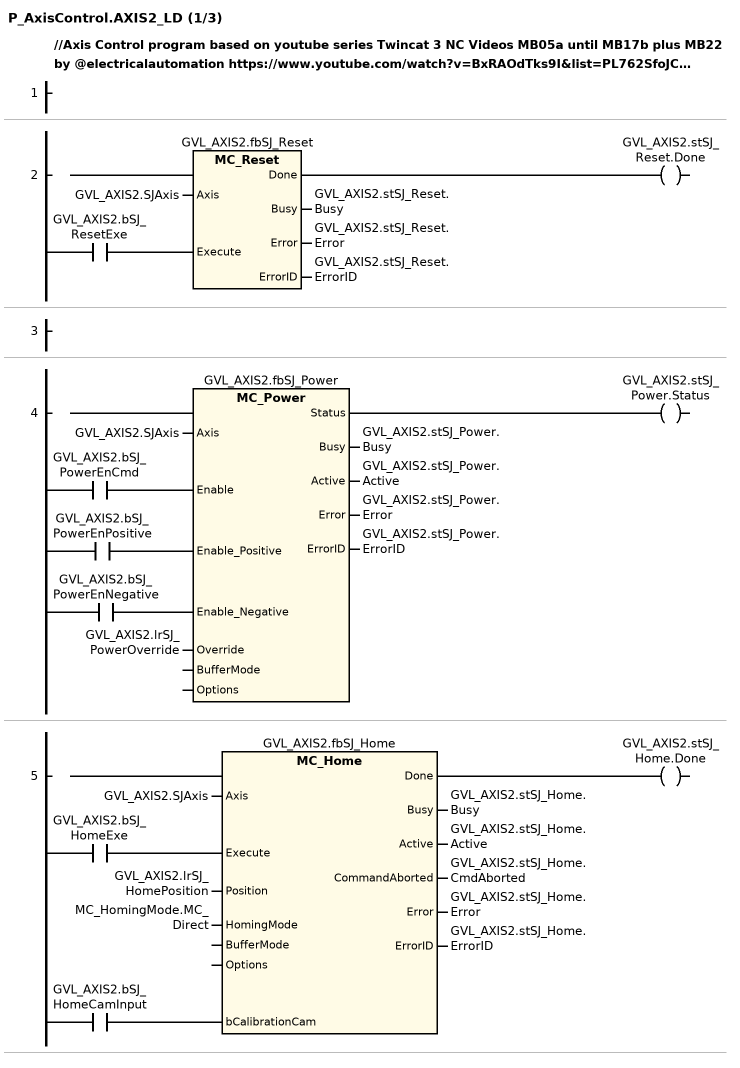
// NETWORK 1: //Axis Control program based on youtube series Twincat 3 NC Videos MB05a until MB17b plus MB22 by @electricalautomation https://www.youtube.com/watch?v=BxRAOdTks9I&list=PL762SfoJC-e8NbAUQ-H7a_TOdqrlBPCw4&index=25

// NETWORK 2
GVL_AXIS2.fbSJ_Reset(
    Axis := GVL_AXIS2.SJAxis,
    Execute := GVL_AXIS2.bSJ_ResetExe,
    Busy => GVL_AXIS2.stSJ_Reset.Busy,
    Error => GVL_AXIS2.stSJ_Reset.Error,
    ErrorID => GVL_AXIS2.stSJ_Reset.ErrorID); // MC_Reset
GVL_AXIS2.stSJ_Reset.Done := GVL_AXIS2.fbSJ_Reset.Done;

// NETWORK 3

// NETWORK 4
GVL_AXIS2.fbSJ_Power(
    Axis := GVL_AXIS2.SJAxis,
    Enable := GVL_AXIS2.bSJ_PowerEnCmd,
    Enable_Positive := GVL_AXIS2.bSJ_PowerEnPositive,
    Enable_Negative := GVL_AXIS2.bSJ_PowerEnNegative,
    Override := GVL_AXIS2.lrSJ_PowerOverride,
    Busy => GVL_AXIS2.stSJ_Power.Busy,
    Active => GVL_AXIS2.stSJ_Power.Active,
    Error => GVL_AXIS2.stSJ_Power.Error,
    ErrorID => GVL_AXIS2.stSJ_Power.ErrorID); // MC_Power
GVL_AXIS2.stSJ_Power.Status := GVL_AXIS2.fbSJ_Power.Status;

// NETWORK 5
GVL_AXIS2.fbSJ_Home(
    Axis := GVL_AXIS2.SJAxis,
    Execute := GVL_AXIS2.bSJ_HomeExe,
    Position := GVL_AXIS2.lrSJ_HomePosition,
    HomingMode := MC_HomingMode.MC_Direct,
    bCalibrationCam := GVL_AXIS2.bSJ_HomeCamInput,
    Busy => GVL_AXIS2.stSJ_Home.Busy,
    Active => GVL_AXIS2.stSJ_Home.Active,
    CommandAborted => GVL_AXIS2.stSJ_Home.CmdAborted,
    Error => GVL_AXIS2.stSJ_Home.Error,
    ErrorID => GVL_AXIS2.stSJ_Home.ErrorID); // MC_Home
GVL_AXIS2.stSJ_Home.Done := GVL_AXIS2.fbSJ_Home.Done;

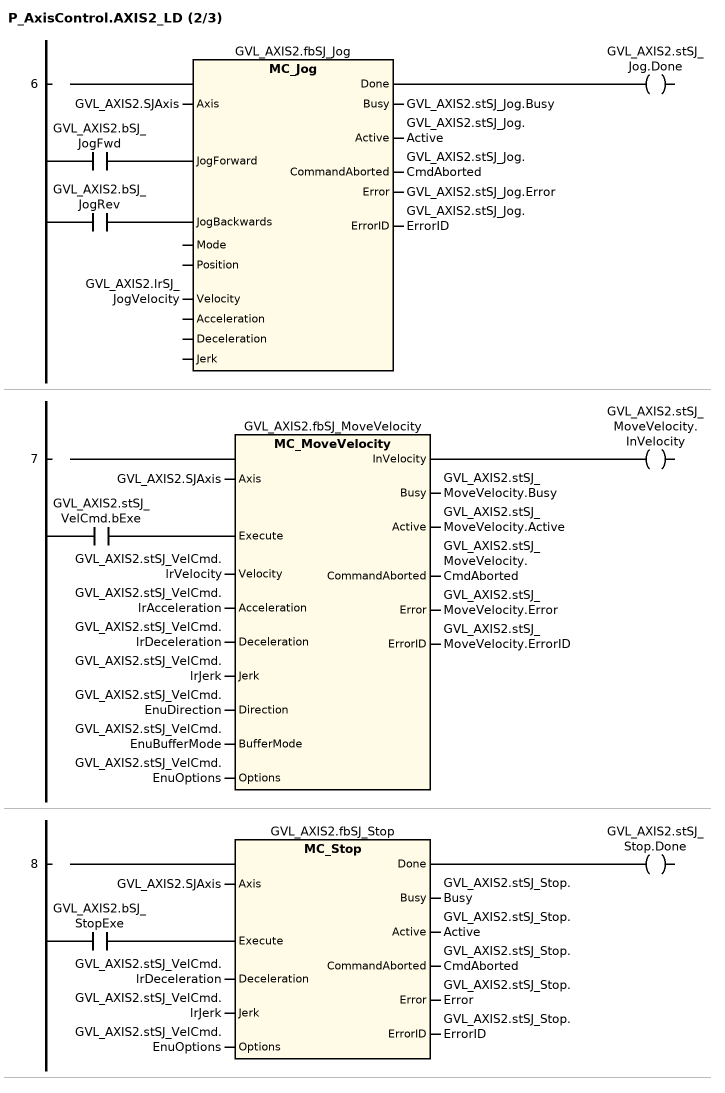
// NETWORK 6
GVL_AXIS2.fbSJ_Jog(
    Axis := GVL_AXIS2.SJAxis,
    JogForward := GVL_AXIS2.bSJ_JogFwd,
    JogBackwards := GVL_AXIS2.bSJ_JogRev,
    Velocity := GVL_AXIS2.lrSJ_JogVelocity,
    Busy => GVL_AXIS2.stSJ_Jog.Busy,
    Active => GVL_AXIS2.stSJ_Jog.Active,
    CommandAborted => GVL_AXIS2.stSJ_Jog.CmdAborted,
    Error => GVL_AXIS2.stSJ_Jog.Error,
    ErrorID => GVL_AXIS2.stSJ_Jog.ErrorID); // MC_Jog
GVL_AXIS2.stSJ_Jog.Done := GVL_AXIS2.fbSJ_Jog.Done;

// NETWORK 7
GVL_AXIS2.fbSJ_MoveVelocity(
    Axis := GVL_AXIS2.SJAxis,
    Execute := GVL_AXIS2.stSJ_VelCmd.bExe,
    Velocity := GVL_AXIS2.stSJ_VelCmd.lrVelocity,
    Acceleration := GVL_AXIS2.stSJ_VelCmd.lrAcceleration,
    Deceleration := GVL_AXIS2.stSJ_VelCmd.lrDeceleration,
    Jerk := GVL_AXIS2.stSJ_VelCmd.lrJerk,
    Direction := GVL_AXIS2.stSJ_VelCmd.EnuDirection,
    BufferMode := GVL_AXIS2.stSJ_VelCmd.EnuBufferMode,
    Options := GVL_AXIS2.stSJ_VelCmd.EnuOptions,
    Busy => GVL_AXIS2.stSJ_MoveVelocity.Busy,
    Active => GVL_AXIS2.stSJ_MoveVelocity.Active,
    CommandAborted => GVL_AXIS2.stSJ_MoveVelocity.CmdAborted,
    Error => GVL_AXIS2.stSJ_MoveVelocity.Error,
    ErrorID => GVL_AXIS2.stSJ_MoveVelocity.ErrorID); // MC_MoveVelocity
GVL_AXIS2.stSJ_MoveVelocity.InVelocity := GVL_AXIS2.fbSJ_MoveVelocity.InVelocity;

// NETWORK 8
GVL_AXIS2.fbSJ_Stop(
    Axis := GVL_AXIS2.SJAxis,
    Execute := GVL_AXIS2.bSJ_StopExe,
    Deceleration := GVL_AXIS2.stSJ_VelCmd.lrDeceleration,
    Jerk := GVL_AXIS2.stSJ_VelCmd.lrJerk,
    Options := GVL_AXIS2.stSJ_VelCmd.EnuOptions,
    Busy => GVL_AXIS2.stSJ_Stop.Busy,
    Active => GVL_AXIS2.stSJ_Stop.Active,
    CommandAborted => GVL_AXIS2.stSJ_Stop.CmdAborted,
    Error => GVL_AXIS2.stSJ_Stop.Error,
    ErrorID => GVL_AXIS2.stSJ_Stop.ErrorID); // MC_Stop
GVL_AXIS2.stSJ_Stop.Done := GVL_AXIS2.fbSJ_Stop.Done;

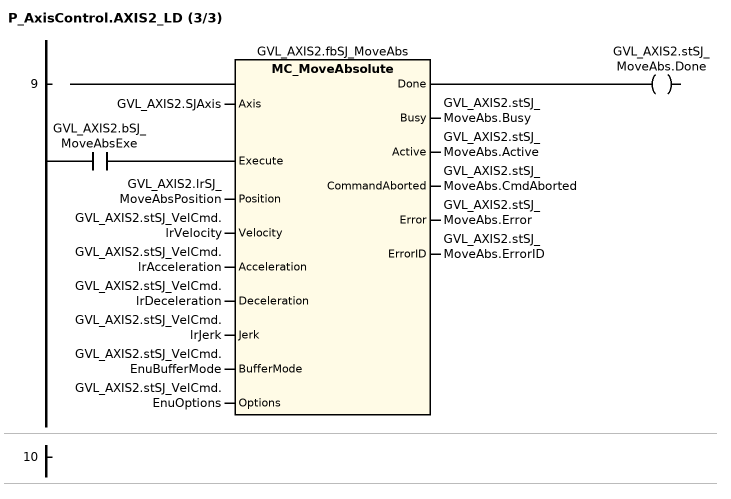
// NETWORK 9
GVL_AXIS2.fbSJ_MoveAbs(
    Axis := GVL_AXIS2.SJAxis,
    Execute := GVL_AXIS2.bSJ_MoveAbsExe,
    Position := GVL_AXIS2.lrSJ_MoveAbsPosition,
    Velocity := GVL_AXIS2.stSJ_VelCmd.lrVelocity,
    Acceleration := GVL_AXIS2.stSJ_VelCmd.lrAcceleration,
    Deceleration := GVL_AXIS2.stSJ_VelCmd.lrDeceleration,
    Jerk := GVL_AXIS2.stSJ_VelCmd.lrJerk,
    BufferMode := GVL_AXIS2.stSJ_VelCmd.EnuBufferMode,
    Options := GVL_AXIS2.stSJ_VelCmd.EnuOptions,
    Busy => GVL_AXIS2.stSJ_MoveAbs.Busy,
    Active => GVL_AXIS2.stSJ_MoveAbs.Active,
    CommandAborted => GVL_AXIS2.stSJ_MoveAbs.CmdAborted,
    Error => GVL_AXIS2.stSJ_MoveAbs.Error,
    ErrorID => GVL_AXIS2.stSJ_MoveAbs.ErrorID); // MC_MoveAbsolute
GVL_AXIS2.stSJ_MoveAbs.Done := GVL_AXIS2.fbSJ_MoveAbs.Done;

// NETWORK 10
END_METHOD

METHOD AXIS3_LD : BOOL
VAR_INPUT
END_VAR
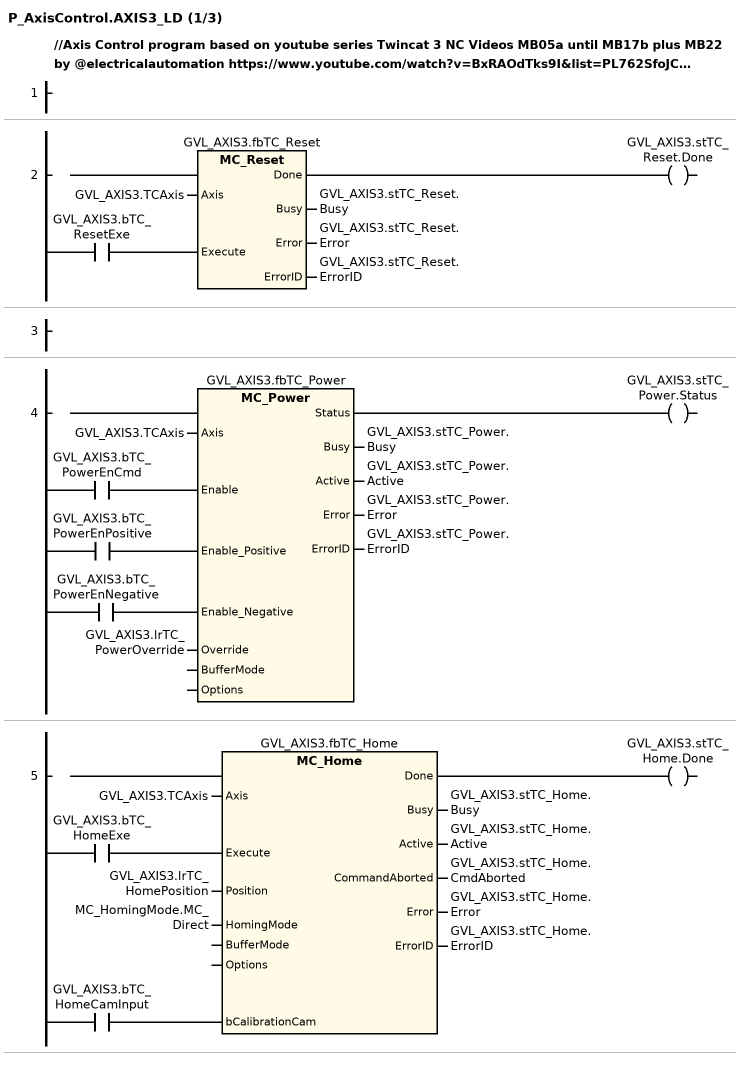
// NETWORK 1: //Axis Control program based on youtube series Twincat 3 NC Videos MB05a until MB17b plus MB22 by @electricalautomation https://www.youtube.com/watch?v=BxRAOdTks9I&list=PL762SfoJC-e8NbAUQ-H7a_TOdqrlBPCw4&index=25

// NETWORK 2
GVL_AXIS3.fbTC_Reset(
    Axis := GVL_AXIS3.TCAxis,
    Execute := GVL_AXIS3.bTC_ResetExe,
    Busy => GVL_AXIS3.stTC_Reset.Busy,
    Error => GVL_AXIS3.stTC_Reset.Error,
    ErrorID => GVL_AXIS3.stTC_Reset.ErrorID); // MC_Reset
GVL_AXIS3.stTC_Reset.Done := GVL_AXIS3.fbTC_Reset.Done;

// NETWORK 3

// NETWORK 4
GVL_AXIS3.fbTC_Power(
    Axis := GVL_AXIS3.TCAxis,
    Enable := GVL_AXIS3.bTC_PowerEnCmd,
    Enable_Positive := GVL_AXIS3.bTC_PowerEnPositive,
    Enable_Negative := GVL_AXIS3.bTC_PowerEnNegative,
    Override := GVL_AXIS3.lrTC_PowerOverride,
    Busy => GVL_AXIS3.stTC_Power.Busy,
    Active => GVL_AXIS3.stTC_Power.Active,
    Error => GVL_AXIS3.stTC_Power.Error,
    ErrorID => GVL_AXIS3.stTC_Power.ErrorID); // MC_Power
GVL_AXIS3.stTC_Power.Status := GVL_AXIS3.fbTC_Power.Status;

// NETWORK 5
GVL_AXIS3.fbTC_Home(
    Axis := GVL_AXIS3.TCAxis,
    Execute := GVL_AXIS3.bTC_HomeExe,
    Position := GVL_AXIS3.lrTC_HomePosition,
    HomingMode := MC_HomingMode.MC_Direct,
    bCalibrationCam := GVL_AXIS3.bTC_HomeCamInput,
    Busy => GVL_AXIS3.stTC_Home.Busy,
    Active => GVL_AXIS3.stTC_Home.Active,
    CommandAborted => GVL_AXIS3.stTC_Home.CmdAborted,
    Error => GVL_AXIS3.stTC_Home.Error,
    ErrorID => GVL_AXIS3.stTC_Home.ErrorID); // MC_Home
GVL_AXIS3.stTC_Home.Done := GVL_AXIS3.fbTC_Home.Done;

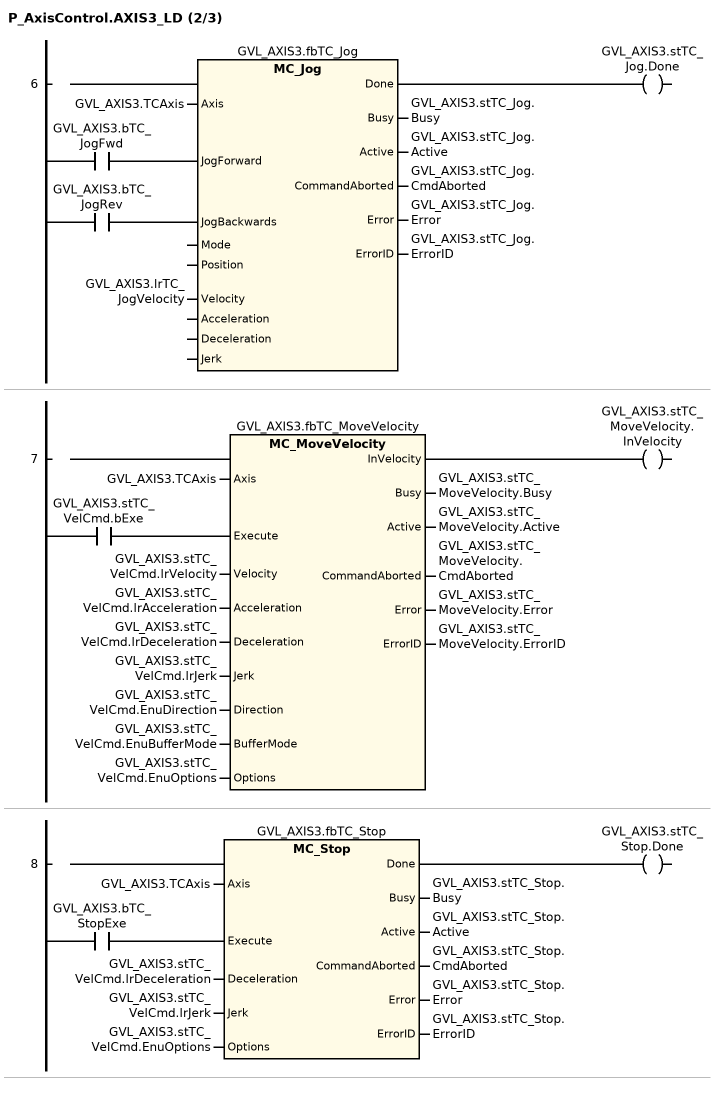
// NETWORK 6
GVL_AXIS3.fbTC_Jog(
    Axis := GVL_AXIS3.TCAxis,
    JogForward := GVL_AXIS3.bTC_JogFwd,
    JogBackwards := GVL_AXIS3.bTC_JogRev,
    Velocity := GVL_AXIS3.lrTC_JogVelocity,
    Busy => GVL_AXIS3.stTC_Jog.Busy,
    Active => GVL_AXIS3.stTC_Jog.Active,
    CommandAborted => GVL_AXIS3.stTC_Jog.CmdAborted,
    Error => GVL_AXIS3.stTC_Jog.Error,
    ErrorID => GVL_AXIS3.stTC_Jog.ErrorID); // MC_Jog
GVL_AXIS3.stTC_Jog.Done := GVL_AXIS3.fbTC_Jog.Done;

// NETWORK 7
GVL_AXIS3.fbTC_MoveVelocity(
    Axis := GVL_AXIS3.TCAxis,
    Execute := GVL_AXIS3.stTC_VelCmd.bExe,
    Velocity := GVL_AXIS3.stTC_VelCmd.lrVelocity,
    Acceleration := GVL_AXIS3.stTC_VelCmd.lrAcceleration,
    Deceleration := GVL_AXIS3.stTC_VelCmd.lrDeceleration,
    Jerk := GVL_AXIS3.stTC_VelCmd.lrJerk,
    Direction := GVL_AXIS3.stTC_VelCmd.EnuDirection,
    BufferMode := GVL_AXIS3.stTC_VelCmd.EnuBufferMode,
    Options := GVL_AXIS3.stTC_VelCmd.EnuOptions,
    Busy => GVL_AXIS3.stTC_MoveVelocity.Busy,
    Active => GVL_AXIS3.stTC_MoveVelocity.Active,
    CommandAborted => GVL_AXIS3.stTC_MoveVelocity.CmdAborted,
    Error => GVL_AXIS3.stTC_MoveVelocity.Error,
    ErrorID => GVL_AXIS3.stTC_MoveVelocity.ErrorID); // MC_MoveVelocity
GVL_AXIS3.stTC_MoveVelocity.InVelocity := GVL_AXIS3.fbTC_MoveVelocity.InVelocity;

// NETWORK 8
GVL_AXIS3.fbTC_Stop(
    Axis := GVL_AXIS3.TCAxis,
    Execute := GVL_AXIS3.bTC_StopExe,
    Deceleration := GVL_AXIS3.stTC_VelCmd.lrDeceleration,
    Jerk := GVL_AXIS3.stTC_VelCmd.lrJerk,
    Options := GVL_AXIS3.stTC_VelCmd.EnuOptions,
    Busy => GVL_AXIS3.stTC_Stop.Busy,
    Active => GVL_AXIS3.stTC_Stop.Active,
    CommandAborted => GVL_AXIS3.stTC_Stop.CmdAborted,
    Error => GVL_AXIS3.stTC_Stop.Error,
    ErrorID => GVL_AXIS3.stTC_Stop.ErrorID); // MC_Stop
GVL_AXIS3.stTC_Stop.Done := GVL_AXIS3.fbTC_Stop.Done;

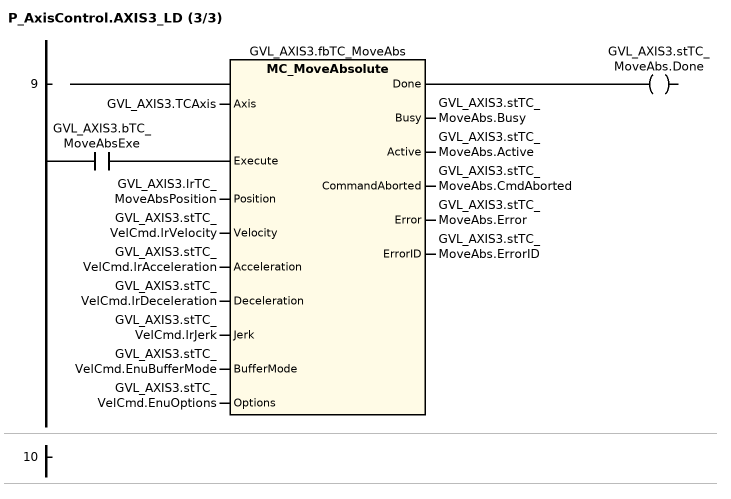
// NETWORK 9
GVL_AXIS3.fbTC_MoveAbs(
    Axis := GVL_AXIS3.TCAxis,
    Execute := GVL_AXIS3.bTC_MoveAbsExe,
    Position := GVL_AXIS3.lrTC_MoveAbsPosition,
    Velocity := GVL_AXIS3.stTC_VelCmd.lrVelocity,
    Acceleration := GVL_AXIS3.stTC_VelCmd.lrAcceleration,
    Deceleration := GVL_AXIS3.stTC_VelCmd.lrDeceleration,
    Jerk := GVL_AXIS3.stTC_VelCmd.lrJerk,
    BufferMode := GVL_AXIS3.stTC_VelCmd.EnuBufferMode,
    Options := GVL_AXIS3.stTC_VelCmd.EnuOptions,
    Busy => GVL_AXIS3.stTC_MoveAbs.Busy,
    Active => GVL_AXIS3.stTC_MoveAbs.Active,
    CommandAborted => GVL_AXIS3.stTC_MoveAbs.CmdAborted,
    Error => GVL_AXIS3.stTC_MoveAbs.Error,
    ErrorID => GVL_AXIS3.stTC_MoveAbs.ErrorID); // MC_MoveAbsolute
GVL_AXIS3.stTC_MoveAbs.Done := GVL_AXIS3.fbTC_MoveAbs.Done;

// NETWORK 10
END_METHOD

METHOD AXIS4_LD : BOOL
VAR_INPUT
END_VAR
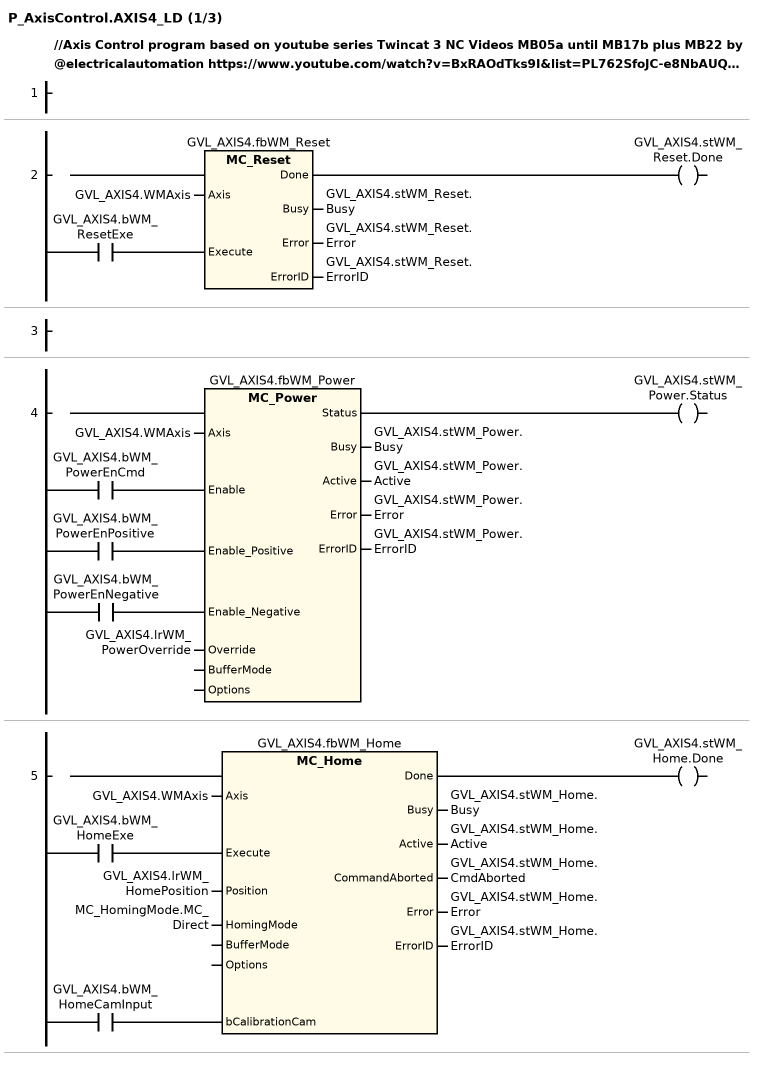
// NETWORK 1: //Axis Control program based on youtube series Twincat 3 NC Videos MB05a until MB17b plus MB22 by @electricalautomation https://www.youtube.com/watch?v=BxRAOdTks9I&list=PL762SfoJC-e8NbAUQ-H7a_TOdqrlBPCw4&index=25

// NETWORK 2
GVL_AXIS4.fbWM_Reset(
    Axis := GVL_AXIS4.WMAxis,
    Execute := GVL_AXIS4.bWM_ResetExe,
    Busy => GVL_AXIS4.stWM_Reset.Busy,
    Error => GVL_AXIS4.stWM_Reset.Error,
    ErrorID => GVL_AXIS4.stWM_Reset.ErrorID); // MC_Reset
GVL_AXIS4.stWM_Reset.Done := GVL_AXIS4.fbWM_Reset.Done;

// NETWORK 3

// NETWORK 4
GVL_AXIS4.fbWM_Power(
    Axis := GVL_AXIS4.WMAxis,
    Enable := GVL_AXIS4.bWM_PowerEnCmd,
    Enable_Positive := GVL_AXIS4.bWM_PowerEnPositive,
    Enable_Negative := GVL_AXIS4.bWM_PowerEnNegative,
    Override := GVL_AXIS4.lrWM_PowerOverride,
    Busy => GVL_AXIS4.stWM_Power.Busy,
    Active => GVL_AXIS4.stWM_Power.Active,
    Error => GVL_AXIS4.stWM_Power.Error,
    ErrorID => GVL_AXIS4.stWM_Power.ErrorID); // MC_Power
GVL_AXIS4.stWM_Power.Status := GVL_AXIS4.fbWM_Power.Status;

// NETWORK 5
GVL_AXIS4.fbWM_Home(
    Axis := GVL_AXIS4.WMAxis,
    Execute := GVL_AXIS4.bWM_HomeExe,
    Position := GVL_AXIS4.lrWM_HomePosition,
    HomingMode := MC_HomingMode.MC_Direct,
    bCalibrationCam := GVL_AXIS4.bWM_HomeCamInput,
    Busy => GVL_AXIS4.stWM_Home.Busy,
    Active => GVL_AXIS4.stWM_Home.Active,
    CommandAborted => GVL_AXIS4.stWM_Home.CmdAborted,
    Error => GVL_AXIS4.stWM_Home.Error,
    ErrorID => GVL_AXIS4.stWM_Home.ErrorID); // MC_Home
GVL_AXIS4.stWM_Home.Done := GVL_AXIS4.fbWM_Home.Done;

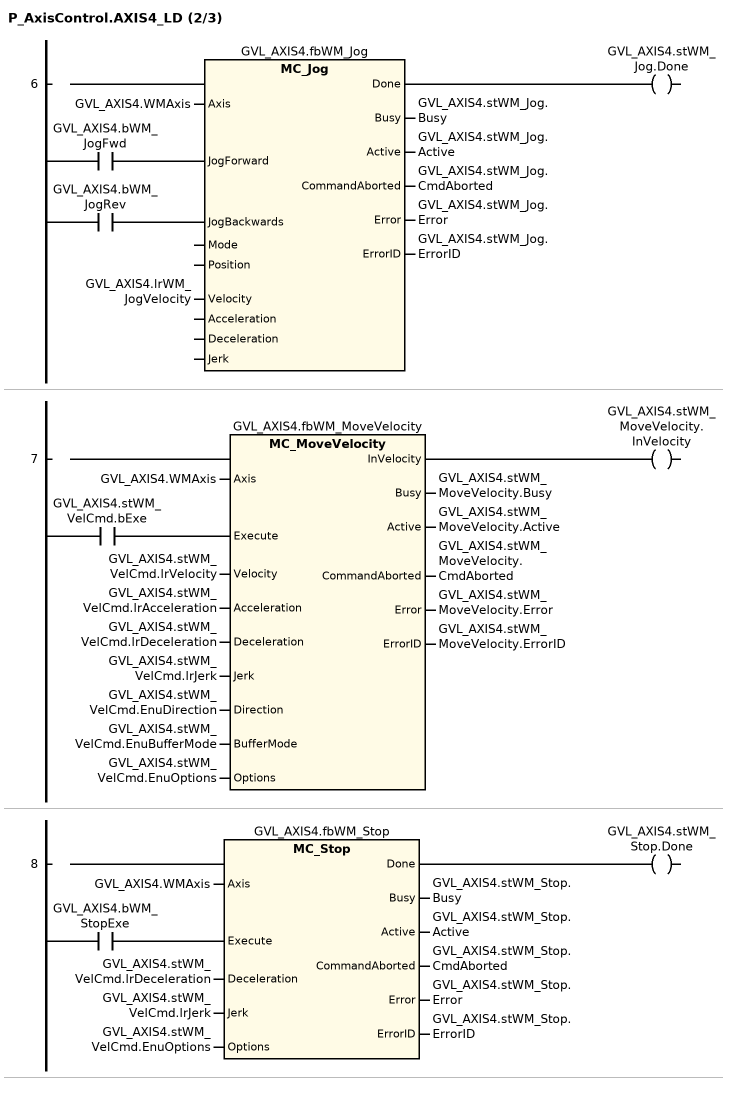
// NETWORK 6
GVL_AXIS4.fbWM_Jog(
    Axis := GVL_AXIS4.WMAxis,
    JogForward := GVL_AXIS4.bWM_JogFwd,
    JogBackwards := GVL_AXIS4.bWM_JogRev,
    Velocity := GVL_AXIS4.lrWM_JogVelocity,
    Busy => GVL_AXIS4.stWM_Jog.Busy,
    Active => GVL_AXIS4.stWM_Jog.Active,
    CommandAborted => GVL_AXIS4.stWM_Jog.CmdAborted,
    Error => GVL_AXIS4.stWM_Jog.Error,
    ErrorID => GVL_AXIS4.stWM_Jog.ErrorID); // MC_Jog
GVL_AXIS4.stWM_Jog.Done := GVL_AXIS4.fbWM_Jog.Done;

// NETWORK 7
GVL_AXIS4.fbWM_MoveVelocity(
    Axis := GVL_AXIS4.WMAxis,
    Execute := GVL_AXIS4.stWM_VelCmd.bExe,
    Velocity := GVL_AXIS4.stWM_VelCmd.lrVelocity,
    Acceleration := GVL_AXIS4.stWM_VelCmd.lrAcceleration,
    Deceleration := GVL_AXIS4.stWM_VelCmd.lrDeceleration,
    Jerk := GVL_AXIS4.stWM_VelCmd.lrJerk,
    Direction := GVL_AXIS4.stWM_VelCmd.EnuDirection,
    BufferMode := GVL_AXIS4.stWM_VelCmd.EnuBufferMode,
    Options := GVL_AXIS4.stWM_VelCmd.EnuOptions,
    Busy => GVL_AXIS4.stWM_MoveVelocity.Busy,
    Active => GVL_AXIS4.stWM_MoveVelocity.Active,
    CommandAborted => GVL_AXIS4.stWM_MoveVelocity.CmdAborted,
    Error => GVL_AXIS4.stWM_MoveVelocity.Error,
    ErrorID => GVL_AXIS4.stWM_MoveVelocity.ErrorID); // MC_MoveVelocity
GVL_AXIS4.stWM_MoveVelocity.InVelocity := GVL_AXIS4.fbWM_MoveVelocity.InVelocity;

// NETWORK 8
GVL_AXIS4.fbWM_Stop(
    Axis := GVL_AXIS4.WMAxis,
    Execute := GVL_AXIS4.bWM_StopExe,
    Deceleration := GVL_AXIS4.stWM_VelCmd.lrDeceleration,
    Jerk := GVL_AXIS4.stWM_VelCmd.lrJerk,
    Options := GVL_AXIS4.stWM_VelCmd.EnuOptions,
    Busy => GVL_AXIS4.stWM_Stop.Busy,
    Active => GVL_AXIS4.stWM_Stop.Active,
    CommandAborted => GVL_AXIS4.stWM_Stop.CmdAborted,
    Error => GVL_AXIS4.stWM_Stop.Error,
    ErrorID => GVL_AXIS4.stWM_Stop.ErrorID); // MC_Stop
GVL_AXIS4.stWM_Stop.Done := GVL_AXIS4.fbWM_Stop.Done;

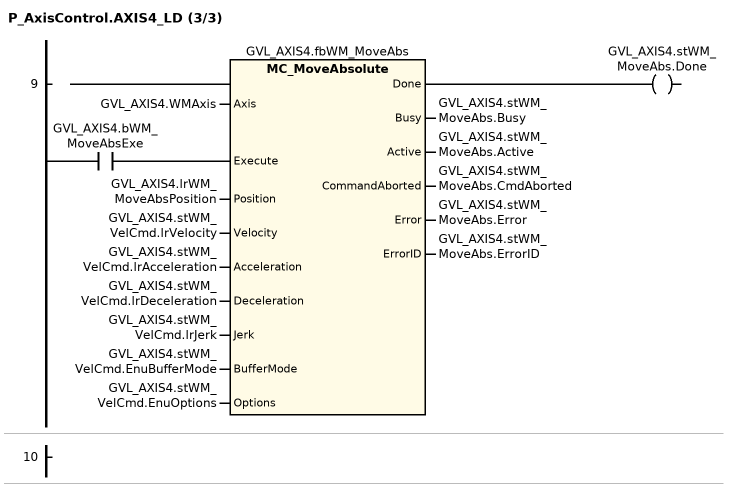
// NETWORK 9
GVL_AXIS4.fbWM_MoveAbs(
    Axis := GVL_AXIS4.WMAxis,
    Execute := GVL_AXIS4.bWM_MoveAbsExe,
    Position := GVL_AXIS4.lrWM_MoveAbsPosition,
    Velocity := GVL_AXIS4.stWM_VelCmd.lrVelocity,
    Acceleration := GVL_AXIS4.stWM_VelCmd.lrAcceleration,
    Deceleration := GVL_AXIS4.stWM_VelCmd.lrDeceleration,
    Jerk := GVL_AXIS4.stWM_VelCmd.lrJerk,
    BufferMode := GVL_AXIS4.stWM_VelCmd.EnuBufferMode,
    Options := GVL_AXIS4.stWM_VelCmd.EnuOptions,
    Busy => GVL_AXIS4.stWM_MoveAbs.Busy,
    Active => GVL_AXIS4.stWM_MoveAbs.Active,
    CommandAborted => GVL_AXIS4.stWM_MoveAbs.CmdAborted,
    Error => GVL_AXIS4.stWM_MoveAbs.Error,
    ErrorID => GVL_AXIS4.stWM_MoveAbs.ErrorID); // MC_MoveAbsolute
GVL_AXIS4.stWM_MoveAbs.Done := GVL_AXIS4.fbWM_MoveAbs.Done;

// NETWORK 10
END_METHOD

END_PROGRAM

// ---- INPUTS/Function Blocks/FB_AnalogInputScaling.TcPOU
FUNCTION_BLOCK FB_AnalogInputScaling
VAR_INPUT
	nRawInput 				: INT;
	stAnalogInputScaling    : ST_AnalogInputScaling;
END_VAR
VAR_OUTPUT
	fOutput 				: LREAL;
END_VAR
VAR
	fRawInput 				: LREAL;
	fNormalizedInput		: LREAL;
END_VAR

fRawInput := INT_TO_LREAL(nRawInput);

fNormalizedInput := (fRawInput - stAnalogInputScaling.fMinInputValue) / (stAnalogInputScaling.fMaxInputValue - stAnalogInputScaling.fMinInputValue);

fOutput := LIMIT(stAnalogInputScaling.fMinOutputValue, stAnalogInputScaling.fMinOutputValue + fNormalizedInput*(stAnalogInputScaling.fMaxOutputValue - stAnalogInputScaling.fMinOutputValue), stAnalogInputScaling.fMaxOutputValue);

END_FUNCTION_BLOCK

// ---- INPUTS/Function Blocks/FB_JoystickInputScaling.TcPOU
FUNCTION_BLOCK FB_JoystickInputScaling
VAR_INPUT
	bEnable  : BOOL;
	nRawInput : INT;
	stJoystickInputScaling : ST_JoystickInputScaling;
END_VAR
VAR_OUTPUT
	fNormalizedOutput : LREAL;
END_VAR
VAR
	fRawInput : LREAL;
	fTempInput : LREAL;
	fTempOutput : LREAL;
END_VAR

fRawInput := INT_TO_REAL(nRawInput);

fTempInput := fRawInput - stJoystickInputScaling.fNeutralInputValue;

IF fTempInput > stJoystickInputScaling.fNeutralDeadband THEN
	fTempOutput := fTempInput/(stJoystickInputScaling.fMaxInputValue - stJoystickInputScaling.fNeutralInputValue);
ELSIF fTempInput < -stJoystickInputScaling.fNeutralDeadband THEN
	fTempOutput := fTempInput/(stJoystickInputScaling.fNeutralInputValue - stJoystickInputScaling.fMinInputValue);
ELSE
	fTempOutput := 0.0;
END_IF
	
IF NOT (bEnable) THEN
	fNormalizedOutput := 0.0;
ELSE 
	fNormalizedOutput := LIMIT(stJoystickInputScaling.fMinOutputValue, fTempOutput, stJoystickInputScaling.fMaxOutputValue);
END_IF

END_FUNCTION_BLOCK

// ---- MACHINE CONTROL/InverseKinematics2d/rt_floord.TcPOU
FUNCTION rt_floord : LREAL
VAR_INPUT
	u: LREAL;
END_VAR
VAR
END_VAR


rt_floord := DINT_TO_LREAL(TRUNC(u));

IF u = rt_floord THEN 
    rt_floord := u;
ELSIF u < 0.0 THEN 
    rt_floord := rt_floord - 1.0;
END_IF;

END_FUNCTION
